		! Move gantry
		MoveAbsJ joints_end, v100, fine, tool0;

		! Read ending positions
		tcp_end_wobj0 := CRobT(\Tool:=tool0\WObj:=wobj0);
		tcp_end_floor := CRobT(\Tool:=tool0\WObj:=WobjFloor);

		TPWrite "End - Gantry: M1=" + NumToStr(joints_end.extax.eax_a, 1) + " M2=" + NumToStr(joints_end.extax.eax_b, 1) + " M3=" + NumToStr(joints_end.extax.eax_c, 1);

		! Calculate TCP changes
		wobj0_dx := tcp_end_wobj0.trans.x - tcp_start_wobj0.trans.x;
		wobj0_dy := tcp_end_wobj0.trans.y - tcp_start_wobj0.trans.y;
		wobj0_dz := tcp_end_wobj0.trans.z - tcp_start_wobj0.trans.z;

		floor_dx := tcp_end_floor.trans.x - tcp_start_floor.trans.x;
		floor_dy := tcp_end_floor.trans.y - tcp_start_floor.trans.y;
		floor_dz := tcp_end_floor.trans.z - tcp_start_floor.trans.z;

		! Save to file
		Open "HOME:/task2_gantry_test.txt", logfile \Append;
		Write logfile, "========================================";
		Write logfile, "TASK2 - Gantry Axis Movement Test (v1.4.0)";
		Write logfile, "Date: " + CDate() + " " + CTime();
		Write logfile, "========================================";
		WaitTime 0.05;
		Write logfile, "Gantry Joint Movement: M1=" + NumToStr(delta_m1, 1) + "mm, M2=" + NumToStr(delta_m2, 1) + "mm, M3=" + NumToStr(delta_m3, 1) + "mm";
		WaitTime 0.05;
		Write logfile, "wobj0 TCP moved: [" + NumToStr(wobj0_dx, 3) + ", " + NumToStr(wobj0_dy, 3) + ", " + NumToStr(wobj0_dz, 3) + "] mm";
		WaitTime 0.05;
		Write logfile, "Floor TCP moved: [" + NumToStr(floor_dx, 3) + ", " + NumToStr(floor_dy, 3) + ", " + NumToStr(floor_dz, 3) + "] mm";
		WaitTime 0.05;
		Write logfile, "========================================";
		Close logfile;

		TPWrite "Saved to: task2_gantry_test.txt";
	ENDPROC

	! ========================================
	! Quick Test - Gantry X Axis Movement
	! ========================================
	! Version: v1.4.1
	! Date: 2025-12-23
	! Purpose: Test M1DM3 (Gantry X) +1000mm movement from current position
	PROC TestGantryX()
		TPWrite "TASK2 - Gantry X Axis Test";
		TPWrite "Testing M1DM3 (X axis) +1000mm";
		TestGantryAxisMovement 1000, 0, 0;
		TPWrite "Test complete!";
	ENDPROC

	! ========================================
	! Quick Test - Gantry Y Axis Movement
	! ========================================
	PROC TestGantryY()
		TPWrite "TASK2 - Gantry Y Axis Test";
		TPWrite "Testing M2DM3 (Y axis) +500mm";
		TestGantryAxisMovement 0, 500, 0;
		TPWrite "Test complete!";
	ENDPROC

	! ========================================
	! Quick Test - Gantry Z Axis Movement
	! ========================================
	PROC TestGantryZ()
		TPWrite "TASK2 - Gantry Z Axis Test";
		TPWrite "Testing M3DM3 (Z axis) +200mm";
		TestGantryAxisMovement 0, 0, 200;
		TPWrite "Test complete!";
	ENDPROC

	! ========================================
	! Robot2 TCP Coordinate Test - XYZ Combined with Return
	! ========================================
	! Version: v1.5.0
	! Date: 2025-12-24
	! Purpose: Move Robot2 TCP in [X+50, Y+30, Z+20] from home position and return
	! MODE Selection (from /HOME/config.txt):
	!   MODE=0 (User's coordinate system):
	!     - Base: WobjFloor
	!     - Floor [+50, +30, +20] -> wobj0 [+50, +30, +20], Floor [+50, +30, +20]
	!   MODE=1 (Claude's coordinate system):
	!     - Base: wobj0
	!     - wobj0 [+50, +30, +20] -> Floor [+50, -30, -20]
	! Changes from v1.4.7:
	!   - Added config.txt MODE support
	!   - MODE=0: Use WobjFloor as base coordinate
	!   - MODE=1: Use wobj0 as base coordinate (default behavior)
	PROC TestRobot2_XYZ()
		VAR jointtarget original_pos;
		VAR jointtarget home_pos;
		VAR num config_mode;

		TPWrite "TASK2 - Robot2 Coordinate Test (v1.5.0)";

		! Read config mode
		config_mode := ReadConfigMode();
		TPWrite "Config MODE=" + NumToStr(config_mode, 0);

		! Save original joint position
		original_pos := CJointT();
		TPWrite "Original joint position saved";

		! Create home position (Robot2: [+90,0,0,0,30,0], keep gantry position)
		home_pos := original_pos;
		home_pos.robax.rax_1 := 90;
		home_pos.robax.rax_2 := 0;
		home_pos.robax.rax_3 := 0;
		home_pos.robax.rax_4 := 0;
		home_pos.robax.rax_5 := 30;
		home_pos.robax.rax_6 := 0;

		! Move to home position
		TPWrite "Moving to home position [+90,0,0,0,30,0]...";
		MoveAbsJ home_pos, v100, fine, tool0;
		TPWrite "At home position";

		! Perform coordinate test based on MODE
		IF config_mode = 0 THEN
			! MODE=0: User's coordinate - use WobjFloor as base
			TPWrite "MODE=0: Moving Floor: [+50, +30, +20]";
			TestCoordinateMovement 50, 30, 20, 0;
		ELSE
			! MODE=1: Claude's coordinate - use wobj0 as base
			TPWrite "MODE=1: Moving wobj0: [+50, +30, +20]";
			TestCoordinateMovement 50, 30, 20, 1;
		ENDIF

		! Return to original joint position
		TPWrite "Returning to original position...";
		MoveAbsJ original_pos, v100, fine, tool0;
		TPWrite "Returned to original position";

		TPWrite "Test complete! Check txt file";
	ENDPROC

	! ========================================
	! Update Robot1 Floor Position (local)
	! ========================================
	! Version: v1.5.2
	! Date: 2025-12-25
	! Purpose: Read Robot1 TCP from T_ROB1 without cross-task procedure call
	PROC UpdateRobot1FloorPositionLocal()
		robot1_floor_pos_t2 := CRobT(\TaskName:="T_ROB1"\Tool:=tool0\WObj:=WobjFloor);
	ENDPROC

	! ========================================
	! Set Robot2 Initial Position
	! ========================================
	! Version: v1.8.7
	! Date: 2026-01-05
	! Purpose: Move Robot2 to initial test position TCP [0, 488, -1000]
	! Position at R-axis center for easy calculation and verification
	! Uses WobjGantry_Rob2 which tracks current gantry position from TASK1
	! Changes in v1.8.7:
	!   - Use gantry extax from TASK1 when issuing MoveJ/MoveL targets
	! NOTE: This procedure does NOT control gantry (only TASK1 can control gantry)
	! Gantry should already be at HOME [0,0,0,0] by TASK1->SetRobot1InitialPosition
	! Version: v1.8.9
	! Date: 2026-01-05
	! Changes in v1.8.9:
	!   - Reduced TPWrite output and file logging to lower 41617 risk
	PROC SetRobot2InitialPosition()
		VAR jointtarget initial_joint;
		VAR jointtarget gantry_joint;
		VAR iodev logfile;

		! Open log file (summary logging)
		Open "HOME:/robot2_init_position.txt", logfile \Write;
		Write logfile, "Robot2 Init (" + TASK2_VERSION + ") Date=" + CDate() + " Time=" + CTime();

		! Step 1: Move Robot2 joints to intermediate position (tWeld2 HOME config)
		TPWrite "Robot2 init: Step1";
		initial_joint := CJointT();
		! Joint angles taught for tWeld2 HOME (confdata [0,0,0,4])
		initial_joint.robax.rax_1 := 0;
		initial_joint.robax.rax_2 := -48.88;
		initial_joint.robax.rax_3 := 6.22;
		initial_joint.robax.rax_4 := 0;
		initial_joint.robax.rax_5 := 8.26;
		initial_joint.robax.rax_6 := 0;
		! Keep current gantry position (DO NOT modify extax!)
		! extax values already set by CJointT()
		MoveAbsJ initial_joint, v100, fine, tool0;
		TPWrite "Robot2 init: Step1 done";
		Write logfile, "Step1 done (intermediate joint)";

		! v1.9.46: Step2 Cartesian refinement REMOVED
		! Robot2 is NOT gantry-configured - controller thinks base is fixed
		! At non-home gantry (especially R!=0), any Cartesian motion (MoveL/MoveJ)
		! converts WobjGantry_Rob2 target to world coords using fixed base -> 50050
		! Step1 MoveAbsJ already sets exact HOME joints - no refinement needed
		! Joint-space motion is gantry-position-independent (always works)

		! Log gantry position for reference
		gantry_joint := CJointT(\TaskName:="T_ROB1");
		Write logfile, "GantryPos from TASK1: X=" + NumToStr(gantry_joint.extax.eax_a,1)
			+ " Y=" + NumToStr(gantry_joint.extax.eax_b,1)
			+ " Z=" + NumToStr(gantry_joint.extax.eax_c,1)
			+ " R=" + NumToStr(gantry_joint.extax.eax_d,1);

		! Log current joint angles for verification
		initial_joint := CJointT();
		Write logfile, "Final joints: J1=" + NumToStr(initial_joint.robax.rax_1, 2)
			+ " J2=" + NumToStr(initial_joint.robax.rax_2, 2)
			+ " J3=" + NumToStr(initial_joint.robax.rax_3, 2)
			+ " J5=" + NumToStr(initial_joint.robax.rax_5, 2);

		TPWrite "Robot2 init: done";
		Write logfile, "Init done (joint-space only) at " + CTime();
		Close logfile;

		! Initialize robot2_floor_pos_t1 for cross-task measurement (v1.7.43)
		UpdateRobot2FloorPosition;
	ERROR
		TPWrite "ERROR in SetRobot2InitialPosition: " + NumToStr(ERRNO, 0);
		Close logfile;
		STOP;
	ENDPROC

	! ========================================
	! Log Current Position (for HOME teaching)
	! ========================================
	! Usage: Jog Robot2 to desired position -> Call from FlexPendant
	!        FlexPendant: ABB Menu -> Program Editor -> Debug -> Call Routine
	! Output: HOME:/current_position_r2.txt
	PROC LogCurrentPosition()
		VAR iodev logfile;
		VAR robtarget rt_tool0;
		VAR robtarget rt_tw2_wobj0;
		VAR robtarget rt_tw2_gantry;
		VAR jointtarget jt;

		Open "HOME:/current_position_r2.txt", logfile \Write;
		Write logfile, "=== ROB_2 Position Log " + CDate() + " " + CTime() + " ===";

		! --- JointTarget ---
		jt := CJointT();
		Write logfile, "";
		Write logfile, "--- ROB_2 JointTarget ---";
		Write logfile, "robax: [" + NumToStr(jt.robax.rax_1,3) + ", "
			+ NumToStr(jt.robax.rax_2,3) + ", " + NumToStr(jt.robax.rax_3,3) + ", "
			+ NumToStr(jt.robax.rax_4,3) + ", " + NumToStr(jt.robax.rax_5,3) + ", "
			+ NumToStr(jt.robax.rax_6,3) + "]";

		! --- RobTarget tool0/wobj0 ---
		rt_tool0 := CRobT(\Tool:=tool0\WObj:=wobj0);
		Write logfile, "";
		Write logfile, "--- ROB_2 RobTarget (tool0, wobj0) ---";
		Write logfile, "[[" + NumToStr(rt_tool0.trans.x,3) + ","
			+ NumToStr(rt_tool0.trans.y,3) + ","
			+ NumToStr(rt_tool0.trans.z,3) + "],["
			+ NumToStr(rt_tool0.rot.q1,5) + ","
			+ NumToStr(rt_tool0.rot.q2,5) + ","
			+ NumToStr(rt_tool0.rot.q3,5) + ","
			+ NumToStr(rt_tool0.rot.q4,5) + "],["
			+ NumToStr(rt_tool0.robconf.cf1,0) + ","
			+ NumToStr(rt_tool0.robconf.cf4,0) + ","
			+ NumToStr(rt_tool0.robconf.cf6,0) + ","
			+ NumToStr(rt_tool0.robconf.cfx,0) + "],extax]";

		! --- RobTarget tWeld2/wobj0 ---
		rt_tw2_wobj0 := CRobT(\Tool:=tWeld2\WObj:=wobj0);
		Write logfile, "";
		Write logfile, "--- ROB_2 RobTarget (tWeld2, wobj0) ---";
		Write logfile, "[[" + NumToStr(rt_tw2_wobj0.trans.x,3) + ","
			+ NumToStr(rt_tw2_wobj0.trans.y,3) + ","
			+ NumToStr(rt_tw2_wobj0.trans.z,3) + "],["
			+ NumToStr(rt_tw2_wobj0.rot.q1,5) + ","
			+ NumToStr(rt_tw2_wobj0.rot.q2,5) + ","
			+ NumToStr(rt_tw2_wobj0.rot.q3,5) + ","
			+ NumToStr(rt_tw2_wobj0.rot.q4,5) + "],["
			+ NumToStr(rt_tw2_wobj0.robconf.cf1,0) + ","
			+ NumToStr(rt_tw2_wobj0.robconf.cf4,0) + ","
			+ NumToStr(rt_tw2_wobj0.robconf.cf6,0) + ","
			+ NumToStr(rt_tw2_wobj0.robconf.cfx,0) + "],extax]";

		! --- RobTarget tWeld2/WobjGantry_Rob2 ---
		UpdateGantryWobj_Rob2;
		rt_tw2_gantry := CRobT(\Tool:=tWeld2\WObj:=WobjGantry_Rob2);
		Write logfile, "";
		Write logfile, "--- ROB_2 RobTarget (tWeld2, WobjGantry_Rob2) ---";
		Write logfile, "[[" + NumToStr(rt_tw2_gantry.trans.x,3) + ","
			+ NumToStr(rt_tw2_gantry.trans.y,3) + ","
			+ NumToStr(rt_tw2_gantry.trans.z,3) + "],["
			+ NumToStr(rt_tw2_gantry.rot.q1,5) + ","
			+ NumToStr(rt_tw2_gantry.rot.q2,5) + ","
			+ NumToStr(rt_tw2_gantry.rot.q3,5) + ","
			+ NumToStr(rt_tw2_gantry.rot.q4,5) + "],["
			+ NumToStr(rt_tw2_gantry.robconf.cf1,0) + ","
			+ NumToStr(rt_tw2_gantry.robconf.cf4,0) + ","
			+ NumToStr(rt_tw2_gantry.robconf.cf6,0) + ","
			+ NumToStr(rt_tw2_gantry.robconf.cfx,0) + "],extax]";

		Close logfile;
		TPWrite "ROB_2 position saved to HOME:/current_position_r2.txt";
	ENDPROC

	! ========================================
	! Set Robot2 TCP Offset for Mode2
	! ========================================
	! Version: v1.8.12
	! Date: 2026-01-06
	! Purpose: Move Robot2 TCP to offset using WobjGantry_Rob2
	! Changes in v1.8.39:
	!   - Use shared offsets from TASK1 (no config.txt read in TASK2)
	PROC SetRobot2OffsetPosition()
		VAR iodev diagfile;
		VAR jointtarget gantry_joint;
		VAR jointtarget task1_joints;  ! v1.8.69: For reading R angle from TASK1
		VAR jointtarget current_joints;  ! v1.8.70: For saving offset joints
		VAR robtarget offset_tcp;
		VAR num tcp_offset_x;
		VAR num tcp_offset_y;
		VAR num tcp_offset_z;
		VAR num wait_count;
		VAR num r_angle;
		VAR num calc_offset_x;
		VAR num calc_offset_y;

		! v1.8.75: Re-add MoveL for initial offset (50426 error fixed in system config)
		! - Initial call: MoveL to offset position using WobjGantry_Rob2
		! - Reposition call: Skip MoveL (joints maintained)

		Open "HOME:/task2_mode2_offset.txt", diagfile \Write;
		Write diagfile, "Mode2 Offset (" + TASK2_VERSION + ") Date=" + CDate() + " Time=" + CTime();

		IF mode2_r2_reposition_trigger THEN
			! ===== REPOSITION CALL =====
			! Gantry has moved, Robot2 joints stay at offset position (no motion needed)
			Write diagfile, "REPOSITION: Joints maintained (no motion)";
			mode2_r2_reposition_done := TRUE;
			TPWrite "R2: Reposition done (joints maintained)";
		ELSE
			! ===== INITIAL CALL =====
			! Move Robot2 TCP to offset position using MoveL
			Write diagfile, "INITIAL: MoveL to offset position";

			! Read offsets from PERS variables (set by TASK1)
			tcp_offset_x := mode2_r2_offset_x;
			tcp_offset_y := mode2_r2_offset_y;
			tcp_offset_z := mode2_r2_offset_z;
			Write diagfile, "Offsets: X=" + NumToStr(tcp_offset_x, 1) + " Y=" + NumToStr(tcp_offset_y, 1) + " Z=" + NumToStr(tcp_offset_z, 1);

			! Update WobjGantry_Rob2 to current gantry position
			UpdateGantryWobj_Rob2;
			gantry_joint := CJointT(\TaskName:="T_ROB1");
			Write diagfile, "WobjGantry_Rob2 updated, gantry extax read";

			! Calculate target position in WobjGantry_Rob2
			! Robot2 init position: [0, 488, -1000] in WobjGantry_Rob2
			! Offset: tcp_offset_y = -100 means 100mm toward Robot2 base
			! Target: [0, 488 + (-100), -1000] = [0, 388, -1000]
			calc_offset_x := tcp_offset_x;
			calc_offset_y := 488 + tcp_offset_y;  ! 488 + (-100) = 388
			Write diagfile, "Target: X=" + NumToStr(calc_offset_x, 1) + " Y=" + NumToStr(calc_offset_y, 1);

			offset_tcp := [[calc_offset_x, calc_offset_y, -1000 + tcp_offset_z],
			               [0.5, -0.5, -0.5, -0.5], [0, 0, 0, 0], gantry_joint.extax];
			Write diagfile, "Offset TCP: [" + NumToStr(offset_tcp.trans.x, 1) + ", "
			               + NumToStr(offset_tcp.trans.y, 1) + ", "
			               + NumToStr(offset_tcp.trans.z, 1) + "]";

			! MoveL to offset position (at HOME, this works)
			TPWrite "R2: MoveL to offset...";
			MoveL offset_tcp, v100, fine, tool0\WObj:=WobjGantry_Rob2;
			TPWrite "R2: MoveL done";
			Write diagfile, "MoveL completed";

			! Save offset joints for reposition calls
			current_joints := CJointT();
			robot2_offset_joints := current_joints.robax;
			Write diagfile, "Offset joints saved";

			! Note: mode2_r2_initial_offset_done is set in main() after config_ready wait
			! This prevents race condition with TASK1's flag reset
			Write diagfile, "MoveL and joint save complete (flag set by main)";
			TPWrite "R2: Offset position reached";
		ENDIF

		Close diagfile;

	ERROR
		Write diagfile, "ERROR in SetRobot2OffsetPosition: " + NumToStr(ERRNO, 0);
		Close diagfile;
		IF ERRNO = ERR_FILEOPEN THEN
			TPWrite "ERROR: Cannot open log file";
		ELSE
			TPWrite "ERROR in SetRobot2OffsetPosition: " + NumToStr(ERRNO, 0);
		ENDIF
		STOP;
	ENDPROC

	! ========================================
	! Update Robot2 Floor Position
	! ========================================
	! Version: v1.7.50
	! Date: 2025-12-31
	! Purpose: Placeholder - TASK1 calculates Robot2 Floor position
	! TASK1's UpdateRobot2BaseDynamicWobj() calculates robot2_floor_pos_t1 directly
	! TASK2 cannot sense gantry movement, so TASK1 does the calculation:
	!   1. TASK1 reads current gantry position
	!   2. TASK1 calculates Robot2 base Floor position
	!   3. TASK1 reads Robot2 TCP wobj0 using CRobT(\TaskName:="T_ROB2")
	!   4. TASK1 combines: robot2_floor_pos_t1 = base Floor + TCP wobj0
	! This procedure does nothing - robot2_floor_pos_t1 already updated by TASK1
	PROC UpdateRobot2FloorPosition()
		! Do nothing - TASK1's UpdateRobot2BaseDynamicWobj() already updated robot2_floor_pos_t1
		! This procedure kept for backward compatibility
		RETURN;
	ENDPROC

	! ========================================
	! Update Gantry Work Object for Robot2
	! ========================================
	! Version: v1.7.50
	! Date: 2025-12-31
	! Purpose: Update WobjGantry_Rob2 to reflect current gantry position and rotation
	! Robot2 cannot control gantry - must read position from TASK1
	! This allows Robot2 TCP control in Floor coordinates regardless of gantry position
	! R-axis orientation: R=0 means gantry parallel to Y-axis (Floor coordinate)
	! Must be called before using WobjGantry_Rob2 for TCP movements
	PROC UpdateGantryWobj_Rob2()
		VAR jointtarget current_gantry;
		VAR num r_deg;

		! Read current gantry position from TASK1 (Robot2 cannot sense this directly)
		current_gantry := CJointT(\TaskName:="T_ROB1");

		! Update WobjGantry_Rob2 position to current gantry location
		WobjGantry_Rob2.uframe.trans.x := current_gantry.extax.eax_a;
		WobjGantry_Rob2.uframe.trans.y := current_gantry.extax.eax_b;
		WobjGantry_Rob2.uframe.trans.z := current_gantry.extax.eax_c;

		! WobjGantry_Rob2 orientation
		! IMPORTANT: WobjGantry_Rob2 coordinate system is always aligned with World/Floor
		! R-axis rotation affects robot base, NOT work object orientation
		! Robot2 base is physically rotated 90deg, but work object remains aligned with World
		! Keep quaternion as identity (no rotation)
		WobjGantry_Rob2.uframe.rot.q1 := 1;
		WobjGantry_Rob2.uframe.rot.q2 := 0;
		WobjGantry_Rob2.uframe.rot.q3 := 0;
		WobjGantry_Rob2.uframe.rot.q4 := 0;

		r_deg := current_gantry.extax.eax_d;

		TPWrite "WobjGantry_Rob2 updated: [" + NumToStr(current_gantry.extax.eax_a,0) + ", "
		                                    + NumToStr(current_gantry.extax.eax_b,0) + ", "
		                                    + NumToStr(current_gantry.extax.eax_c,0) + ", R="
		                                    + NumToStr(r_deg,1) + "]";
	ENDPROC

	! ========================================
	! Calculate Robot Distance
	! ========================================
	! Version: v1.5.1
	! Date: 2025-12-25
	! Purpose: Calculate 3D distance between Robot1 and Robot2 in Floor coordinate
	! Returns: Distance in mm
	FUNC num CalculateRobotDistance()
		VAR num dx;
		VAR num dy;
		VAR num dz;

		dx := robot2_floor_pos_t1.trans.x - robot1_floor_pos_t2.trans.x;
		dy := robot2_floor_pos_t1.trans.y - robot1_floor_pos_t2.trans.y;
		dz := robot2_floor_pos_t1.trans.z - robot1_floor_pos_t2.trans.z;

		RETURN Sqrt(Pow(dx, 2) + Pow(dy, 2) + Pow(dz, 2));
	ENDFUNC

	! ========================================
	! Measure Robot Distance
	! ========================================
	! Version: v1.5.1
	! Date: 2025-12-25
	! Purpose: Measure and log distance between Robot1 and Robot2
	! Output: TP display + /HOME/robot_distance_log.txt
	PROC MeasureRobotDistance()
		VAR num distance;
		VAR iodev logfile;

		TPWrite "========================================";
		TPWrite "Robot Distance Measurement (v1.5.1)";
		TPWrite "========================================";

		! Update both robot positions
		UpdateRobot1FloorPositionLocal;
		UpdateRobot2FloorPosition;

		! Calculate distance
		distance := CalculateRobotDistance();

		! Display on TP
		TPWrite "Robot1 Floor Position:";
		TPWrite "  X = " + NumToStr(robot1_floor_pos_t2.trans.x, 2) + " mm";
		TPWrite "  Y = " + NumToStr(robot1_floor_pos_t2.trans.y, 2) + " mm";
		TPWrite "  Z = " + NumToStr(robot1_floor_pos_t2.trans.z, 2) + " mm";
		TPWrite "";
		TPWrite "Robot2 Floor Position:";
		TPWrite "  X = " + NumToStr(robot2_floor_pos_t1.trans.x, 2) + " mm";
		TPWrite "  Y = " + NumToStr(robot2_floor_pos_t1.trans.y, 2) + " mm";
		TPWrite "  Z = " + NumToStr(robot2_floor_pos_t1.trans.z, 2) + " mm";
		TPWrite "";
		TPWrite "Distance between robots: " + NumToStr(distance, 2) + " mm";
		TPWrite "========================================";

		! Save to log file
		Open "HOME:/robot_distance_log.txt", logfile \Write;

		Write logfile, "========================================";
		Write logfile, "Robot Distance Measurement (v1.5.1)";
		Write logfile, "========================================";
		Write logfile, "Date: " + CDate();
		Write logfile, "Time: " + CTime();
		Write logfile, "";
		Write logfile, "Robot1 Floor Position (tool0):";
		Write logfile, "  X = " + NumToStr(robot1_floor_pos_t2.trans.x, 2) + " mm";
		Write logfile, "  Y = " + NumToStr(robot1_floor_pos_t2.trans.y, 2) + " mm";
		Write logfile, "  Z = " + NumToStr(robot1_floor_pos_t2.trans.z, 2) + " mm";
		Write logfile, "";
		Write logfile, "Robot2 Floor Position (tool0):";
		Write logfile, "  X = " + NumToStr(robot2_floor_pos_t1.trans.x, 2) + " mm";
		Write logfile, "  Y = " + NumToStr(robot2_floor_pos_t1.trans.y, 2) + " mm";
		Write logfile, "  Z = " + NumToStr(robot2_floor_pos_t1.trans.z, 2) + " mm";
		Write logfile, "";
		Write logfile, "Distance: " + NumToStr(distance, 2) + " mm";
		Write logfile, "========================================\0A";

		Close logfile;
		TPWrite "Saved to: /HOME/robot_distance_log.txt";

	ERROR
		TPWrite "ERROR in MeasureRobotDistance: " + NumToStr(ERRNO, 0);
		Close logfile;
		TRYNEXT;
	ENDPROC

	! ========================================
	! Test Robot2 Base Height
	! ========================================
	! Version: v1.7.14
	! Date: 2025-12-28
	! Purpose: Check tool0 TCP height from base at specific joint angles
	! Uses WobjFloor_Rob2
	! Output: TP display + /HOME/robot2_base_height.txt
	PROC TestRobot2BaseHeight()
		VAR jointtarget test_pos;
		VAR robtarget tcp_wobj0;
		VAR robtarget tcp_floor;
		VAR iodev logfile;

		TPWrite "========================================";
		TPWrite "Robot2 Base Height Test (v1.7.14)";

		! Get current position
		test_pos := CJointT();

		! Set robot joints to [+90, 0, 0, 0, 0, 0]
		test_pos.robax.rax_1 := 90;
		test_pos.robax.rax_2 := 0;
		test_pos.robax.rax_3 := 0;
		test_pos.robax.rax_4 := 0;
		test_pos.robax.rax_5 := 0;
		test_pos.robax.rax_6 := 0;

		! Move to test position
		TPWrite "Moving to test position [+90,0,0,0,0,0]...";
		MoveAbsJ test_pos, v100, fine, tool0;
		WaitTime 0.5;

		! Read TCP position in wobj0
		tcp_wobj0 := CRobT(\Tool:=tool0\WObj:=wobj0);

		! Read TCP position in Floor coordinate (using Robot2-specific Floor)
		tcp_floor := CRobT(\Tool:=tool0\WObj:=WobjFloor_Rob2);

		! Display on TP
		TPWrite "Robot2 wobj0:";
		TPWrite "  X = " + NumToStr(tcp_wobj0.trans.x, 2);
		TPWrite "  Y = " + NumToStr(tcp_wobj0.trans.y, 2);
		TPWrite "  Z = " + NumToStr(tcp_wobj0.trans.z, 2);

		TPWrite "Robot2 Floor (WobjFloor_Rob2):";
		TPWrite "  X = " + NumToStr(tcp_floor.trans.x, 2);
		TPWrite "  Y = " + NumToStr(tcp_floor.trans.y, 2);
		TPWrite "  Z = " + NumToStr(tcp_floor.trans.z, 2);

		TPWrite "========================================";

		! Save to log file
		Open "HOME:/robot2_base_height.txt", logfile \Write;

		Write logfile, "========================================";
		Write logfile, "Robot2 Base Height Test (v1.7.14)";
		Write logfile, "========================================";
		Write logfile, "Date: " + CDate();
		Write logfile, "Time: " + CTime();
		Write logfile, "";
		Write logfile, "Joint Angles: [+90, 0, 0, 0, 0, 0]";
		Write logfile, "";
		Write logfile, "Robot2 wobj0 (tool0):";
		Write logfile, "  X = " + NumToStr(tcp_wobj0.trans.x, 2) + " mm";
		Write logfile, "  Y = " + NumToStr(tcp_wobj0.trans.y, 2) + " mm";
		Write logfile, "  Z = " + NumToStr(tcp_wobj0.trans.z, 2) + " mm";
		Write logfile, "";
		Write logfile, "Robot2 Floor (tool0) - using WobjFloor_Rob2:";
		Write logfile, "  X = " + NumToStr(tcp_floor.trans.x, 2) + " mm";
		Write logfile, "  Y = " + NumToStr(tcp_floor.trans.y, 2) + " mm";
		Write logfile, "  Z = " + NumToStr(tcp_floor.trans.z, 2) + " mm";
		Write logfile, "========================================\0A";

		Close logfile;
		TPWrite "Saved to: /HOME/robot2_base_height.txt";

	ERROR
		TPWrite "ERROR in TestRobot2BaseHeight: " + NumToStr(ERRNO, 0);
		Close logfile;
		TRYNEXT;
	ENDPROC

	! ========================================
	! Test Gantry Movement Effect on Floor Coordinates
	! ========================================
	! Version: v1.7.29
	! Date: 2025-12-29
	! Purpose: Test if Floor coordinates change when gantry moves
	! Reads gantry movement from config.txt (X, Y, Z, R)
	! Initial position: Robot1 [-90,0,0,0,0,0], Robot2 [+90,0,0,0,0,0]
	! Gantry HOME: [-9500, 5300, 700, 0] (safe Z position, max=1000mm)
	! Gantry moved: HOME + config offset
	! Note: Based on 12-23 backup fnCoordToJoint function
	! Output: /HOME/gantry_floor_test.txt
	PROC TestGantryFloorCoordinates()
		VAR jointtarget rob1_init;
		VAR jointtarget rob2_init;
		VAR jointtarget home_pos;
		VAR jointtarget moved_pos;
		VAR robtarget rob1_floor_before;
		VAR robtarget rob2_floor_before;
		VAR robtarget rob1_floor_after;
		VAR robtarget rob2_floor_after;
		VAR iodev logfile;
		VAR iodev configfile;
		VAR string line;
		VAR string value_str;
		VAR bool found_value;
		VAR bool found_x;
		VAR bool found_y;
		VAR bool found_z;
		VAR bool found_r;
		VAR num gantry_x_offset;
		VAR num gantry_y_offset;
		VAR num gantry_z_offset;
		VAR num gantry_r_offset;

		TPWrite "========================================";
		TPWrite "Gantry Floor Test (v1.7.28)";

		! Initialize variables
		gantry_x_offset := 0;
		gantry_y_offset := 0;
		gantry_z_offset := 0;
		gantry_r_offset := 0;

		! Check Robot1 position
		TPWrite "Checking Robot1 position...";
		rob1_init := CJointT(\TaskName:="T_ROB1");
		IF Abs(rob1_init.robax.rax_1 + 90) > 5 THEN
			TPWrite "WARNING: Robot1 is NOT at initial position!";
			TPWrite "Current Robot1 J1: " + NumToStr(rob1_init.robax.rax_1, 1);
			TPWrite "Expected: -90 degrees";
			TPWrite "Please run TASK1->SetRobot1InitialPosition first";
			TPWrite "Then re-run this test";
			STOP;
		ENDIF
		TPWrite "Robot1 position OK (J1=-90)";

		! Move Robot2 to initial test position (keep current gantry position)
		TPWrite "Moving Robot2 to initial position...";
		rob2_init := CJointT();
		! Set robot joints only
		rob2_init.robax.rax_1 := 90;
		rob2_init.robax.rax_2 := 0;
		rob2_init.robax.rax_3 := 0;
		rob2_init.robax.rax_4 := 0;
		rob2_init.robax.rax_5 := 0;
		rob2_init.robax.rax_6 := 0;
		! Keep current gantry position (DO NOT force to 0)
		! extax values already set by CJointT()
		MoveAbsJ rob2_init, v100, fine, tool0;
		TPWrite "Robot2 initial position reached!";

		! Now move gantry to HOME position
		TPWrite "Moving gantry to HOME position...";
		home_pos := rob2_init;
		home_pos.extax.eax_a := -9500;  ! X1 = WobjFloor origin X
		home_pos.extax.eax_b := 5300;   ! Y = WobjFloor origin Y
		home_pos.extax.eax_c := 700;    ! Z = Safe mid-height (max=1000, ref: 12-23 backup)
		home_pos.extax.eax_d := 0;      ! R = 0
		! eax_e: keep from CJointT() (not used)
		home_pos.extax.eax_f := -9500;  ! X2 = X1 (Master-Follower sync!)
		MoveAbsJ home_pos, v100, fine, tool0;
		TPWrite "Gantry at HOME position (WobjFloor origin)";
		TPWrite "Both robots ready!";

		! Read gantry offsets from config.txt (simple approach)
		TPWrite "Opening config.txt...";
		Open "HOME:/config.txt", configfile \Read;
		TPWrite "Reading config values...";

		! Read GANTRY_X
		found_x := FALSE;
		WHILE found_x = FALSE DO
			line := ReadStr(configfile \RemoveCR);
			IF StrFind(line, 1, "GANTRY_X=") = 1 THEN
				IF StrLen(line) >= 10 THEN
					value_str := StrPart(line, 10, StrLen(line) - 9);
					found_value := StrToVal(value_str, gantry_x_offset);
					found_x := TRUE;
					TPWrite "Found GANTRY_X=" + NumToStr(gantry_x_offset, 0);
				ENDIF
			ENDIF
		ENDWHILE

		! Read GANTRY_Y
		found_y := FALSE;
		WHILE found_y = FALSE DO
			line := ReadStr(configfile \RemoveCR);
			IF StrFind(line, 1, "GANTRY_Y=") = 1 THEN
				IF StrLen(line) >= 10 THEN
					value_str := StrPart(line, 10, StrLen(line) - 9);
					found_value := StrToVal(value_str, gantry_y_offset);
					found_y := TRUE;
					TPWrite "Found GANTRY_Y=" + NumToStr(gantry_y_offset, 0);
				ENDIF
			ENDIF
		ENDWHILE

		! Read GANTRY_Z
		found_z := FALSE;
		WHILE found_z = FALSE DO
			line := ReadStr(configfile \RemoveCR);
			IF StrFind(line, 1, "GANTRY_Z=") = 1 THEN
				IF StrLen(line) >= 10 THEN
					value_str := StrPart(line, 10, StrLen(line) - 9);
					found_value := StrToVal(value_str, gantry_z_offset);
					found_z := TRUE;
					TPWrite "Found GANTRY_Z=" + NumToStr(gantry_z_offset, 0);
				ENDIF
			ENDIF
		ENDWHILE

		! Read GANTRY_R
		found_r := FALSE;
		WHILE found_r = FALSE DO
			line := ReadStr(configfile \RemoveCR);
			IF StrFind(line, 1, "GANTRY_R=") = 1 THEN
				IF StrLen(line) >= 10 THEN
					value_str := StrPart(line, 10, StrLen(line) - 9);
					found_value := StrToVal(value_str, gantry_r_offset);
					found_r := TRUE;
					TPWrite "Found GANTRY_R=" + NumToStr(gantry_r_offset, 1);
				ENDIF
			ENDIF
		ENDWHILE

		Close configfile;
		TPWrite "Config reading complete!";

		TPWrite "Gantry offsets:";
		TPWrite "  X=" + NumToStr(gantry_x_offset, 0) + " mm";
		TPWrite "  Y=" + NumToStr(gantry_y_offset, 0) + " mm";
		TPWrite "  Z=" + NumToStr(gantry_z_offset, 0) + " mm";
		TPWrite "  R=" + NumToStr(gantry_r_offset, 1) + " deg";

		! Move to HOME position (all gantry axes = 0)
		TPWrite "Moving to HOME position...";
		home_pos := CJointT();
		home_pos.extax.eax_a := 0;  ! X axis
		home_pos.extax.eax_b := 0;  ! Y axis
		home_pos.extax.eax_c := 0;  ! Z axis
		home_pos.extax.eax_d := 0;  ! R axis
		MoveAbsJ home_pos, v100, fine, tool0;
		WaitTime 1.0;

		! Measure BEFORE gantry movement
		TPWrite "Measuring before gantry move...";
		UpdateRobot1FloorPositionLocal;
		UpdateRobot2FloorPosition;
		rob1_floor_before := robot1_floor_pos_t2;
		rob2_floor_before := robot2_floor_pos_t1;

		! Move gantry axes (HOME + offset)
		TPWrite "Moving gantry...";
		moved_pos := home_pos;
		moved_pos.extax.eax_a := -9500 + gantry_x_offset;  ! X1 = HOME + offset
		moved_pos.extax.eax_b := 5300 + gantry_y_offset;   ! Y = HOME + offset
		moved_pos.extax.eax_c := 700 + gantry_z_offset;    ! Z = HOME + offset (max=1000)
		moved_pos.extax.eax_d := 0 + gantry_r_offset;      ! R = HOME + offset
		! eax_e: keep from home_pos/CJointT() (not used)
		moved_pos.extax.eax_f := -9500 + gantry_x_offset;  ! X2 = X1 (Master-Follower sync!)
		MoveAbsJ moved_pos, v100, fine, tool0;
		WaitTime 1.0;

		! Measure AFTER gantry movement
		TPWrite "Measuring after gantry move...";
		UpdateRobot1FloorPositionLocal;
		UpdateRobot2FloorPosition;
		rob1_floor_after := robot1_floor_pos_t2;
		rob2_floor_after := robot2_floor_pos_t1;

		! Return to HOME position
		TPWrite "Returning to HOME position...";
		MoveAbsJ home_pos, v100, fine, tool0;

		! Save results
		Open "HOME:/gantry_floor_test.txt", logfile \Write;

		Write logfile, "========================================";
		Write logfile, "Gantry Floor Coordinate Test (v1.7.29)";
		Write logfile, "========================================";
		Write logfile, "Date: " + CDate();
		Write logfile, "Time: " + CTime();
		Write logfile, "";
		Write logfile, "HOME Position (WobjFloor origin):";
		Write logfile, "  Gantry: X1=-9500, Y=5300, Z=2100, R=0, X2=-9500";
		Write logfile, "";
		Write logfile, "Initial Position:";
		Write logfile, "  Robot1: [-90,0,0,0,0,0]";
		Write logfile, "  Robot2: [+90,0,0,0,0,0]";
		Write logfile, "  Gantry: at HOME (WobjFloor origin)";
		Write logfile, "";
		Write logfile, "Gantry Movement:";
		Write logfile, "  X = " + NumToStr(gantry_x_offset, 2) + " mm (X1 and X2 synchronized)";
		Write logfile, "  Y = " + NumToStr(gantry_y_offset, 2) + " mm";
		Write logfile, "  Z = " + NumToStr(gantry_z_offset, 2) + " mm";
		Write logfile, "  R = " + NumToStr(gantry_r_offset, 2) + " deg";
		Write logfile, "";
		Write logfile, "BEFORE Gantry Movement:";
		Write logfile, "------------------------";
		Write logfile, "Robot1 Floor (tool0):";
		Write logfile, "  X = " + NumToStr(rob1_floor_before.trans.x, 2) + " mm";
		Write logfile, "  Y = " + NumToStr(rob1_floor_before.trans.y, 2) + " mm";
		Write logfile, "  Z = " + NumToStr(rob1_floor_before.trans.z, 2) + " mm";
		Write logfile, "";
		Write logfile, "Robot2 Floor (tool0):";
		Write logfile, "  X = " + NumToStr(rob2_floor_before.trans.x, 2) + " mm";
		Write logfile, "  Y = " + NumToStr(rob2_floor_before.trans.y, 2) + " mm";
		Write logfile, "  Z = " + NumToStr(rob2_floor_before.trans.z, 2) + " mm";
		Write logfile, "";
		Write logfile, "AFTER Gantry Movement:";
		Write logfile, "----------------------";
		Write logfile, "Robot1 Floor (tool0):";
		Write logfile, "  X = " + NumToStr(rob1_floor_after.trans.x, 2) + " mm";
		Write logfile, "  Y = " + NumToStr(rob1_floor_after.trans.y, 2) + " mm";
		Write logfile, "  Z = " + NumToStr(rob1_floor_after.trans.z, 2) + " mm";
		Write logfile, "";
		Write logfile, "Robot2 Floor (tool0):";
		Write logfile, "  X = " + NumToStr(rob2_floor_after.trans.x, 2) + " mm";
		Write logfile, "  Y = " + NumToStr(rob2_floor_after.trans.y, 2) + " mm";
		Write logfile, "  Z = " + NumToStr(rob2_floor_after.trans.z, 2) + " mm";
		Write logfile, "";
		Write logfile, "DIFFERENCE:";
		Write logfile, "-----------";
		Write logfile, "Robot1 Floor Delta:";
		Write logfile, "  dX = " + NumToStr(rob1_floor_after.trans.x - rob1_floor_before.trans.x, 2) + " mm";
		Write logfile, "  dY = " + NumToStr(rob1_floor_after.trans.y - rob1_floor_before.trans.y, 2) + " mm";
		Write logfile, "  dZ = " + NumToStr(rob1_floor_after.trans.z - rob1_floor_before.trans.z, 2) + " mm";
		Write logfile, "";
		Write logfile, "Robot2 Floor Delta:";
		Write logfile, "  dX = " + NumToStr(rob2_floor_after.trans.x - rob2_floor_before.trans.x, 2) + " mm";
		Write logfile, "  dY = " + NumToStr(rob2_floor_after.trans.y - rob2_floor_before.trans.y, 2) + " mm";
		Write logfile, "  dZ = " + NumToStr(rob2_floor_after.trans.z - rob2_floor_before.trans.z, 2) + " mm";
		Write logfile, "========================================\0A";

		Close logfile;
		TPWrite "Saved to: /HOME/gantry_floor_test.txt";
		TPWrite "Test complete!";

	ERROR
		IF ERRNO = ERR_FILEOPEN THEN
			TPWrite "ERROR: Cannot open config.txt";
			STOP;
		ELSEIF ERRNO = ERR_FILEACC THEN
			TPWrite "ERROR: End of file or access error";
			TPWrite "Check config.txt format";
			Close configfile;
			STOP;
		ELSE
			TPWrite "ERROR in TestGantryFloorCoordinates";
			TPWrite "ERRNO: " + NumToStr(ERRNO, 0);
			Close logfile;
			Close configfile;
			STOP;
		ENDIF
	ENDPROC

! ========================================
! Weld Sequence Procedures (v1.9.0)
! ========================================
! Purpose: Robot2 weld sequence synchronization with TASK1
! Robot2 waits for TASK1 signal, then moves to weld position

! ----------------------------------------
! Robot2 Weld Ready - Wait and Move (2-step approach)
! ----------------------------------------
! v1.9.19: Step1 - MoveAbsJ to safe joint position
!          Step2 - MoveJ to wobj0 target position
PROC Robot2_WeldReady()
	VAR robtarget weld_target;
	VAR jointtarget safe_jt;

	TPWrite "[R2_WELD] Robot2 weld ready procedure started";
	TPWrite "[R2_WELD] Waiting for TASK1 weld start signal...";

	! Wait for TASK1 weld start signal
	WHILE NOT t1_weld_start DO
		WaitTime 0.1;
	ENDWHILE

	TPWrite "[R2_WELD] Received weld start signal from TASK1";

	! Step 1: Move to safe JOINT position first
	! Robot joints: [0, -10, -50, 0, -30, 0]
	safe_jt := CJointT();
	safe_jt.robax.rax_1 := 0;
	safe_jt.robax.rax_2 := -10;
	safe_jt.robax.rax_3 := -50;
	safe_jt.robax.rax_4 := 0;
	safe_jt.robax.rax_5 := -30;
	safe_jt.robax.rax_6 := 0;
	! Robot2 has no external axes
	safe_jt.extax.eax_a := 9E9;
	safe_jt.extax.eax_b := 9E9;
	safe_jt.extax.eax_c := 9E9;
	safe_jt.extax.eax_d := 9E9;
	safe_jt.extax.eax_e := 9E9;
	safe_jt.extax.eax_f := 9E9;
	TPWrite "[R2_WELD] Step1: MoveAbsJ to safe joints";
	MoveAbsJ safe_jt, v100, fine, tool0;

	! Step 2: Move to wobj0 target position
	! wobj0 target: [0, 118, -1300]
	weld_target.trans.x := 0;
	weld_target.trans.y := 118;
	weld_target.trans.z := -1300;
	weld_target.rot.q1 := WELD_R2_ORIENT_Q1;
	weld_target.rot.q2 := WELD_R2_ORIENT_Q2;
	weld_target.rot.q3 := WELD_R2_ORIENT_Q3;
	weld_target.rot.q4 := WELD_R2_ORIENT_Q4;
	weld_target.robconf.cf1 := 0;
	weld_target.robconf.cf4 := 0;
	weld_target.robconf.cf6 := 0;
	weld_target.robconf.cfx := 0;
	weld_target.extax.eax_a := 9E9;
	weld_target.extax.eax_b := 9E9;
	weld_target.extax.eax_c := 9E9;
	weld_target.extax.eax_d := 9E9;
	weld_target.extax.eax_e := 9E9;
	weld_target.extax.eax_f := 9E9;

	TPWrite "[R2_WELD] Step2: MoveJ to wobj0 [0, 118, -1300]";
	MoveJ weld_target, v100, fine, tool0\WObj:=wobj0;

	! Signal ready to TASK1
	t2_weld_ready := TRUE;

	TPWrite "[R2_WELD] Robot2 at weld position, signaled ready";
ENDPROC

! ----------------------------------------
! Robot2 Weld Hold - Maintain Position
! ----------------------------------------
! Maintains weld posture while TASK1 moves gantry
! Called after Robot2_WeldReady completes
PROC Robot2_WeldHold()
	TPWrite "[R2_WELD] Robot2 holding weld position...";

	! Wait for TASK1 weld complete signal
	WHILE NOT t1_weld_done DO
		WaitTime 0.1;
	ENDWHILE

	TPWrite "[R2_WELD] TASK1 weld complete, Robot2 released";
ENDPROC

! ----------------------------------------
! Robot2 Weld Sequence (Combined)
! ----------------------------------------
! Combined sequence: wait for signal, move to position, hold until done
PROC Robot2_WeldSequence()
	TPWrite "========================================";
	TPWrite "[R2_WELD] v1.9.0 Robot2 Weld Sequence Start";
	TPWrite "========================================";

	! Reset ready flag
	t2_weld_ready := FALSE;

	! Wait for signal and move to weld position
	Robot2_WeldReady;

	! Hold position until welding complete
	Robot2_WeldHold;

	TPWrite "========================================";
	TPWrite "[R2_WELD] Robot2 Weld Sequence Complete!";
	TPWrite "========================================";
ENDPROC

! ========================================
! Edge-based Weld Sequence (v2.0.0)
! ========================================
! Ported from PlanA - waits for TASK1 to position gantry,
! then moves Robot2 to weld position considering bRobSwap

! ----------------------------------------
! Robot2 Edge-based Weld Sequence (v1.9.37)
! ----------------------------------------
! Waits for t1_weld_position_ready, then positions Robot2
! v1.9.37: Weld tracking with position logging, edge data from TASK1
PROC Robot2_EdgeWeldSequence()
    ! ========================================
    ! Robot2 Edge Weld Sequence (v3.0.0)
    ! Ported from PlanA rWeld012()
    ! Uses Welds2{} + wobjWeldLine2 + fCalcWeldingpos()
    ! Simulation mode: MoveL (WELD_ARC_ENABLED=FALSE)
    ! ========================================
    VAR num nTempMmps;
    VAR num nHoldWeldVel;
    VAR jointtarget jCurrent;
    VAR iodev weld2_errlog;
    VAR num nErrorCount;
    VAR num nMotionErrorCount;

    TPWrite "[R2_WELD] Robot2_EdgeWeldSequence v4.0 start";
    nHoldWeldVel:=0.01;

    ! Signal TASK1 we are ready (unblocks Step 7 wait in Full Weld Sequence)
    t2_weld_ready := TRUE;

    ! --- Setup weld data (wd1..wd40) ---
    wd1:=[Welds2{1}.cpm/6,0,[5,0,Welds2{1}.voltage,Welds2{1}.wfs,0,Welds2{1}.Current,0,0,0],[0,0,0,0,0,0,0,0,0]];
    wd2:=[Welds2{2}.cpm/6,0,[5,0,Welds2{2}.voltage,Welds2{2}.wfs,0,Welds2{2}.Current,0,0,0],[0,0,0,0,0,0,0,0,0]];
    wd3:=[Welds2{3}.cpm/6,0,[5,0,Welds2{3}.voltage,Welds2{3}.wfs,0,Welds2{3}.Current,0,0,0],[0,0,0,0,0,0,0,0,0]];
    wd4:=[Welds2{4}.cpm/6,0,[5,0,Welds2{4}.voltage,Welds2{4}.wfs,0,Welds2{4}.Current,0,0,0],[0,0,0,0,0,0,0,0,0]];
    wd5:=[Welds2{5}.cpm/6,0,[5,0,Welds2{5}.voltage,Welds2{5}.wfs,0,Welds2{5}.Current,0,0,0],[0,0,0,0,0,0,0,0,0]];
    wd6:=[Welds2{6}.cpm/6,0,[5,0,Welds2{6}.voltage,Welds2{6}.wfs,0,Welds2{6}.Current,0,0,0],[0,0,0,0,0,0,0,0,0]];
    wd7:=[Welds2{7}.cpm/6,0,[5,0,Welds2{7}.voltage,Welds2{7}.wfs,0,Welds2{7}.Current,0,0,0],[0,0,0,0,0,0,0,0,0]];
    wd8:=[Welds2{8}.cpm/6,0,[5,0,Welds2{8}.voltage,Welds2{8}.wfs,0,Welds2{8}.Current,0,0,0],[0,0,0,0,0,0,0,0,0]];
    wd9:=[Welds2{9}.cpm/6,0,[5,0,Welds2{9}.voltage,Welds2{9}.wfs,0,Welds2{9}.Current,0,0,0],[0,0,0,0,0,0,0,0,0]];
    wd10:=[Welds2{10}.cpm/6,0,[5,0,Welds2{10}.voltage,Welds2{10}.wfs,0,Welds2{10}.Current,0,0,0],[0,0,0,0,0,0,0,0,0]];
    wd11:=[Welds2{11}.cpm/6,0,[5,0,Welds2{11}.voltage,Welds2{11}.wfs,0,Welds2{11}.Current,0,0,0],[0,0,0,0,0,0,0,0,0]];
    wd12:=[Welds2{12}.cpm/6,0,[5,0,Welds2{12}.voltage,Welds2{12}.wfs,0,Welds2{12}.Current,0,0,0],[0,0,0,0,0,0,0,0,0]];
    wd13:=[Welds2{13}.cpm/6,0,[5,0,Welds2{13}.voltage,Welds2{13}.wfs,0,Welds2{13}.Current,0,0,0],[0,0,0,0,0,0,0,0,0]];
    wd14:=[Welds2{14}.cpm/6,0,[5,0,Welds2{14}.voltage,Welds2{14}.wfs,0,Welds2{14}.Current,0,0,0],[0,0,0,0,0,0,0,0,0]];
    wd15:=[Welds2{15}.cpm/6,0,[5,0,Welds2{15}.voltage,Welds2{15}.wfs,0,Welds2{15}.Current,0,0,0],[0,0,0,0,0,0,0,0,0]];
    wd16:=[Welds2{16}.cpm/6,0,[5,0,Welds2{16}.voltage,Welds2{16}.wfs,0,Welds2{16}.Current,0,0,0],[0,0,0,0,0,0,0,0,0]];
    wd17:=[Welds2{17}.cpm/6,0,[5,0,Welds2{17}.voltage,Welds2{17}.wfs,0,Welds2{17}.Current,0,0,0],[0,0,0,0,0,0,0,0,0]];
    wd18:=[Welds2{18}.cpm/6,0,[5,0,Welds2{18}.voltage,Welds2{18}.wfs,0,Welds2{18}.Current,0,0,0],[0,0,0,0,0,0,0,0,0]];
    wd19:=[Welds2{19}.cpm/6,0,[5,0,Welds2{19}.voltage,Welds2{19}.wfs,0,Welds2{19}.Current,0,0,0],[0,0,0,0,0,0,0,0,0]];
    wd20:=[Welds2{20}.cpm/6,0,[5,0,Welds2{20}.voltage,Welds2{20}.wfs,0,Welds2{20}.Current,0,0,0],[0,0,0,0,0,0,0,0,0]];
    wd21:=[Welds2{21}.cpm/6,0,[5,0,Welds2{21}.voltage,Welds2{21}.wfs,0,Welds2{21}.Current,0,0,0],[0,0,0,0,0,0,0,0,0]];
    wd22:=[Welds2{22}.cpm/6,0,[5,0,Welds2{22}.voltage,Welds2{22}.wfs,0,Welds2{22}.Current,0,0,0],[0,0,0,0,0,0,0,0,0]];
    wd23:=[Welds2{23}.cpm/6,0,[5,0,Welds2{23}.voltage,Welds2{23}.wfs,0,Welds2{23}.Current,0,0,0],[0,0,0,0,0,0,0,0,0]];
    wd24:=[Welds2{24}.cpm/6,0,[5,0,Welds2{24}.voltage,Welds2{24}.wfs,0,Welds2{24}.Current,0,0,0],[0,0,0,0,0,0,0,0,0]];
    wd25:=[Welds2{25}.cpm/6,0,[5,0,Welds2{25}.voltage,Welds2{25}.wfs,0,Welds2{25}.Current,0,0,0],[0,0,0,0,0,0,0,0,0]];
    wd26:=[Welds2{26}.cpm/6,0,[5,0,Welds2{26}.voltage,Welds2{26}.wfs,0,Welds2{26}.Current,0,0,0],[0,0,0,0,0,0,0,0,0]];
    wd27:=[Welds2{27}.cpm/6,0,[5,0,Welds2{27}.voltage,Welds2{27}.wfs,0,Welds2{27}.Current,0,0,0],[0,0,0,0,0,0,0,0,0]];
    wd28:=[Welds2{28}.cpm/6,0,[5,0,Welds2{28}.voltage,Welds2{28}.wfs,0,Welds2{28}.Current,0,0,0],[0,0,0,0,0,0,0,0,0]];
    wd29:=[Welds2{29}.cpm/6,0,[5,0,Welds2{29}.voltage,Welds2{29}.wfs,0,Welds2{29}.Current,0,0,0],[0,0,0,0,0,0,0,0,0]];
    wd30:=[Welds2{30}.cpm/6,0,[5,0,Welds2{30}.voltage,Welds2{30}.wfs,0,Welds2{30}.Current,0,0,0],[0,0,0,0,0,0,0,0,0]];
    wd31:=[Welds2{31}.cpm/6,0,[5,0,Welds2{31}.voltage,Welds2{31}.wfs,0,Welds2{31}.Current,0,0,0],[0,0,0,0,0,0,0,0,0]];
    wd32:=[Welds2{32}.cpm/6,0,[5,0,Welds2{32}.voltage,Welds2{32}.wfs,0,Welds2{32}.Current,0,0,0],[0,0,0,0,0,0,0,0,0]];
    wd33:=[Welds2{33}.cpm/6,0,[5,0,Welds2{33}.voltage,Welds2{33}.wfs,0,Welds2{33}.Current,0,0,0],[0,0,0,0,0,0,0,0,0]];
    wd34:=[Welds2{34}.cpm/6,0,[5,0,Welds2{34}.voltage,Welds2{34}.wfs,0,Welds2{34}.Current,0,0,0],[0,0,0,0,0,0,0,0,0]];
    wd35:=[Welds2{35}.cpm/6,0,[5,0,Welds2{35}.voltage,Welds2{35}.wfs,0,Welds2{35}.Current,0,0,0],[0,0,0,0,0,0,0,0,0]];
    wd36:=[Welds2{36}.cpm/6,0,[5,0,Welds2{36}.voltage,Welds2{36}.wfs,0,Welds2{36}.Current,0,0,0],[0,0,0,0,0,0,0,0,0]];
    wd37:=[Welds2{37}.cpm/6,0,[5,0,Welds2{37}.voltage,Welds2{37}.wfs,0,Welds2{37}.Current,0,0,0],[0,0,0,0,0,0,0,0,0]];
    wd38:=[Welds2{38}.cpm/6,0,[5,0,Welds2{38}.voltage,Welds2{38}.wfs,0,Welds2{38}.Current,0,0,0],[0,0,0,0,0,0,0,0,0]];
    wd39:=[Welds2{39}.cpm/6,0,[5,0,Welds2{39}.voltage,Welds2{39}.wfs,0,Welds2{39}.Current,0,0,0],[0,0,0,0,0,0,0,0,0]];
    wd40:=[Welds2{nMotionStepCount{2}}.cpm/6,0,[5,0,Welds2{nMotionStepCount{2}}.voltage,Welds2{nMotionStepCount{2}}.wfs,0,Welds2{nMotionStepCount{2}}.Current,0,0,0],[0,0,0,0,0,0,0,0,0]];

    Holdwd1:=[nHoldWeldVel,0,[5,0,Welds2{1}.voltage,Welds2{1}.wfs,0,Welds2{1}.Current,0,0,0],[0,0,0,0,0,0,0,0,0]];
    Holdwd2:=[nHoldWeldVel,0,[5,0,Welds2{2}.voltage,Welds2{2}.wfs,0,Welds2{2}.Current,0,0,0],[0,0,0,0,0,0,0,0,0]];
    Holdwd3:=[nHoldWeldVel,0,[5,0,Welds2{3}.voltage,Welds2{3}.wfs,0,Welds2{3}.Current,0,0,0],[0,0,0,0,0,0,0,0,0]];
    Holdwd4:=[nHoldWeldVel,0,[5,0,Welds2{4}.voltage,Welds2{4}.wfs,0,Welds2{4}.Current,0,0,0],[0,0,0,0,0,0,0,0,0]];
    Holdwd5:=[nHoldWeldVel,0,[5,0,Welds2{5}.voltage,Welds2{5}.wfs,0,Welds2{5}.Current,0,0,0],[0,0,0,0,0,0,0,0,0]];
    Holdwd6:=[nHoldWeldVel,0,[5,0,Welds2{6}.voltage,Welds2{6}.wfs,0,Welds2{6}.Current,0,0,0],[0,0,0,0,0,0,0,0,0]];
    Holdwd7:=[nHoldWeldVel,0,[5,0,Welds2{7}.voltage,Welds2{7}.wfs,0,Welds2{7}.Current,0,0,0],[0,0,0,0,0,0,0,0,0]];
    Holdwd8:=[nHoldWeldVel,0,[5,0,Welds2{8}.voltage,Welds2{8}.wfs,0,Welds2{8}.Current,0,0,0],[0,0,0,0,0,0,0,0,0]];
    Holdwd9:=[nHoldWeldVel,0,[5,0,Welds2{9}.voltage,Welds2{9}.wfs,0,Welds2{9}.Current,0,0,0],[0,0,0,0,0,0,0,0,0]];
    Holdwd10:=[nHoldWeldVel,0,[5,0,Welds2{10}.voltage,Welds2{10}.wfs,0,Welds2{10}.Current,0,0,0],[0,0,0,0,0,0,0,0,0]];

    ! --- Setup weave data (weave1..weave40) ---
    weave1:=[Welds2{1}.WeaveShape,Welds2{1}.WeaveType,Welds2{1}.WeaveLength,Welds2{1}.WeaveWidth,0,Welds2{1}.WeaveDwellLeft,0,Welds2{1}.WeaveDwellRight,0,0,0,0,0,0,0];
    weave2:=[Welds2{2}.WeaveShape,Welds2{2}.WeaveType,Welds2{2}.WeaveLength,Welds2{2}.WeaveWidth,0,Welds2{2}.WeaveDwellLeft,0,Welds2{2}.WeaveDwellRight,0,0,0,0,0,0,0];
    weave3:=[Welds2{3}.WeaveShape,Welds2{3}.WeaveType,Welds2{3}.WeaveLength,Welds2{3}.WeaveWidth,0,Welds2{3}.WeaveDwellLeft,0,Welds2{3}.WeaveDwellRight,0,0,0,0,0,0,0];
    weave4:=[Welds2{4}.WeaveShape,Welds2{4}.WeaveType,Welds2{4}.WeaveLength,Welds2{4}.WeaveWidth,0,Welds2{4}.WeaveDwellLeft,0,Welds2{4}.WeaveDwellRight,0,0,0,0,0,0,0];
    weave5:=[Welds2{5}.WeaveShape,Welds2{5}.WeaveType,Welds2{5}.WeaveLength,Welds2{5}.WeaveWidth,0,Welds2{5}.WeaveDwellLeft,0,Welds2{5}.WeaveDwellRight,0,0,0,0,0,0,0];
    weave6:=[Welds2{6}.WeaveShape,Welds2{6}.WeaveType,Welds2{6}.WeaveLength,Welds2{6}.WeaveWidth,0,Welds2{6}.WeaveDwellLeft,0,Welds2{6}.WeaveDwellRight,0,0,0,0,0,0,0];
    weave7:=[Welds2{7}.WeaveShape,Welds2{7}.WeaveType,Welds2{7}.WeaveLength,Welds2{7}.WeaveWidth,0,Welds2{7}.WeaveDwellLeft,0,Welds2{7}.WeaveDwellRight,0,0,0,0,0,0,0];
    weave8:=[Welds2{8}.WeaveShape,Welds2{8}.WeaveType,Welds2{8}.WeaveLength,Welds2{8}.WeaveWidth,0,Welds2{8}.WeaveDwellLeft,0,Welds2{8}.WeaveDwellRight,0,0,0,0,0,0,0];
    weave9:=[Welds2{9}.WeaveShape,Welds2{9}.WeaveType,Welds2{9}.WeaveLength,Welds2{9}.WeaveWidth,0,Welds2{9}.WeaveDwellLeft,0,Welds2{9}.WeaveDwellRight,0,0,0,0,0,0,0];
    weave10:=[Welds2{10}.WeaveShape,Welds2{10}.WeaveType,Welds2{10}.WeaveLength,Welds2{10}.WeaveWidth,0,Welds2{10}.WeaveDwellLeft,0,Welds2{10}.WeaveDwellRight,0,0,0,0,0,0,0];
    weave11:=[Welds2{11}.WeaveShape,Welds2{11}.WeaveType,Welds2{11}.WeaveLength,Welds2{11}.WeaveWidth,0,Welds2{11}.WeaveDwellLeft,0,Welds2{11}.WeaveDwellRight,0,0,0,0,0,0,0];
    weave12:=[Welds2{12}.WeaveShape,Welds2{12}.WeaveType,Welds2{12}.WeaveLength,Welds2{12}.WeaveWidth,0,Welds2{12}.WeaveDwellLeft,0,Welds2{12}.WeaveDwellRight,0,0,0,0,0,0,0];
    weave13:=[Welds2{13}.WeaveShape,Welds2{13}.WeaveType,Welds2{13}.WeaveLength,Welds2{13}.WeaveWidth,0,Welds2{13}.WeaveDwellLeft,0,Welds2{13}.WeaveDwellRight,0,0,0,0,0,0,0];
    weave14:=[Welds2{14}.WeaveShape,Welds2{14}.WeaveType,Welds2{14}.WeaveLength,Welds2{14}.WeaveWidth,0,Welds2{14}.WeaveDwellLeft,0,Welds2{14}.WeaveDwellRight,0,0,0,0,0,0,0];
    weave15:=[Welds2{15}.WeaveShape,Welds2{15}.WeaveType,Welds2{15}.WeaveLength,Welds2{15}.WeaveWidth,0,Welds2{15}.WeaveDwellLeft,0,Welds2{15}.WeaveDwellRight,0,0,0,0,0,0,0];
    weave16:=[Welds2{16}.WeaveShape,Welds2{16}.WeaveType,Welds2{16}.WeaveLength,Welds2{16}.WeaveWidth,0,Welds2{16}.WeaveDwellLeft,0,Welds2{16}.WeaveDwellRight,0,0,0,0,0,0,0];
    weave17:=[Welds2{17}.WeaveShape,Welds2{17}.WeaveType,Welds2{17}.WeaveLength,Welds2{17}.WeaveWidth,0,Welds2{17}.WeaveDwellLeft,0,Welds2{17}.WeaveDwellRight,0,0,0,0,0,0,0];
    weave18:=[Welds2{18}.WeaveShape,Welds2{18}.WeaveType,Welds2{18}.WeaveLength,Welds2{18}.WeaveWidth,0,Welds2{18}.WeaveDwellLeft,0,Welds2{18}.WeaveDwellRight,0,0,0,0,0,0,0];
    weave19:=[Welds2{19}.WeaveShape,Welds2{19}.WeaveType,Welds2{19}.WeaveLength,Welds2{19}.WeaveWidth,0,Welds2{19}.WeaveDwellLeft,0,Welds2{19}.WeaveDwellRight,0,0,0,0,0,0,0];
    weave20:=[Welds2{20}.WeaveShape,Welds2{20}.WeaveType,Welds2{20}.WeaveLength,Welds2{20}.WeaveWidth,0,Welds2{20}.WeaveDwellLeft,0,Welds2{20}.WeaveDwellRight,0,0,0,0,0,0,0];
    weave21:=[Welds2{21}.WeaveShape,Welds2{21}.WeaveType,Welds2{21}.WeaveLength,Welds2{21}.WeaveWidth,0,Welds2{21}.WeaveDwellLeft,0,Welds2{21}.WeaveDwellRight,0,0,0,0,0,0,0];
    weave22:=[Welds2{22}.WeaveShape,Welds2{22}.WeaveType,Welds2{22}.WeaveLength,Welds2{22}.WeaveWidth,0,Welds2{22}.WeaveDwellLeft,0,Welds2{22}.WeaveDwellRight,0,0,0,0,0,0,0];
    weave23:=[Welds2{23}.WeaveShape,Welds2{23}.WeaveType,Welds2{23}.WeaveLength,Welds2{23}.WeaveWidth,0,Welds2{23}.WeaveDwellLeft,0,Welds2{23}.WeaveDwellRight,0,0,0,0,0,0,0];
    weave24:=[Welds2{24}.WeaveShape,Welds2{24}.WeaveType,Welds2{24}.WeaveLength,Welds2{24}.WeaveWidth,0,Welds2{24}.WeaveDwellLeft,0,Welds2{24}.WeaveDwellRight,0,0,0,0,0,0,0];
    weave25:=[Welds2{25}.WeaveShape,Welds2{25}.WeaveType,Welds2{25}.WeaveLength,Welds2{25}.WeaveWidth,0,Welds2{25}.WeaveDwellLeft,0,Welds2{25}.WeaveDwellRight,0,0,0,0,0,0,0];
    weave26:=[Welds2{26}.WeaveShape,Welds2{26}.WeaveType,Welds2{26}.WeaveLength,Welds2{26}.WeaveWidth,0,Welds2{26}.WeaveDwellLeft,0,Welds2{26}.WeaveDwellRight,0,0,0,0,0,0,0];
    weave27:=[Welds2{27}.WeaveShape,Welds2{27}.WeaveType,Welds2{27}.WeaveLength,Welds2{27}.WeaveWidth,0,Welds2{27}.WeaveDwellLeft,0,Welds2{27}.WeaveDwellRight,0,0,0,0,0,0,0];
    weave28:=[Welds2{28}.WeaveShape,Welds2{28}.WeaveType,Welds2{28}.WeaveLength,Welds2{28}.WeaveWidth,0,Welds2{28}.WeaveDwellLeft,0,Welds2{28}.WeaveDwellRight,0,0,0,0,0,0,0];
    weave29:=[Welds2{29}.WeaveShape,Welds2{29}.WeaveType,Welds2{29}.WeaveLength,Welds2{29}.WeaveWidth,0,Welds2{29}.WeaveDwellLeft,0,Welds2{29}.WeaveDwellRight,0,0,0,0,0,0,0];
    weave30:=[Welds2{30}.WeaveShape,Welds2{30}.WeaveType,Welds2{30}.WeaveLength,Welds2{30}.WeaveWidth,0,Welds2{30}.WeaveDwellLeft,0,Welds2{30}.WeaveDwellRight,0,0,0,0,0,0,0];
    weave31:=[Welds2{31}.WeaveShape,Welds2{31}.WeaveType,Welds2{31}.WeaveLength,Welds2{31}.WeaveWidth,0,Welds2{31}.WeaveDwellLeft,0,Welds2{31}.WeaveDwellRight,0,0,0,0,0,0,0];
    weave32:=[Welds2{32}.WeaveShape,Welds2{32}.WeaveType,Welds2{32}.WeaveLength,Welds2{32}.WeaveWidth,0,Welds2{32}.WeaveDwellLeft,0,Welds2{32}.WeaveDwellRight,0,0,0,0,0,0,0];
    weave33:=[Welds2{33}.WeaveShape,Welds2{33}.WeaveType,Welds2{33}.WeaveLength,Welds2{33}.WeaveWidth,0,Welds2{33}.WeaveDwellLeft,0,Welds2{33}.WeaveDwellRight,0,0,0,0,0,0,0];
    weave34:=[Welds2{34}.WeaveShape,Welds2{34}.WeaveType,Welds2{34}.WeaveLength,Welds2{34}.WeaveWidth,0,Welds2{34}.WeaveDwellLeft,0,Welds2{34}.WeaveDwellRight,0,0,0,0,0,0,0];
    weave35:=[Welds2{35}.WeaveShape,Welds2{35}.WeaveType,Welds2{35}.WeaveLength,Welds2{35}.WeaveWidth,0,Welds2{35}.WeaveDwellLeft,0,Welds2{35}.WeaveDwellRight,0,0,0,0,0,0,0];
    weave36:=[Welds2{36}.WeaveShape,Welds2{36}.WeaveType,Welds2{36}.WeaveLength,Welds2{36}.WeaveWidth,0,Welds2{36}.WeaveDwellLeft,0,Welds2{36}.WeaveDwellRight,0,0,0,0,0,0,0];
    weave37:=[Welds2{37}.WeaveShape,Welds2{37}.WeaveType,Welds2{37}.WeaveLength,Welds2{37}.WeaveWidth,0,Welds2{37}.WeaveDwellLeft,0,Welds2{37}.WeaveDwellRight,0,0,0,0,0,0,0];
    weave38:=[Welds2{38}.WeaveShape,Welds2{38}.WeaveType,Welds2{38}.WeaveLength,Welds2{38}.WeaveWidth,0,Welds2{38}.WeaveDwellLeft,0,Welds2{38}.WeaveDwellRight,0,0,0,0,0,0,0];
    weave39:=[Welds2{39}.WeaveShape,Welds2{39}.WeaveType,Welds2{39}.WeaveLength,Welds2{39}.WeaveWidth,0,Welds2{39}.WeaveDwellLeft,0,Welds2{39}.WeaveDwellRight,0,0,0,0,0,0,0];
    weave40:=[Welds2{nMotionStepCount{2}}.WeaveShape,Welds2{nMotionStepCount{2}}.WeaveType,Welds2{nMotionStepCount{2}}.WeaveLength,Welds2{nMotionStepCount{2}}.WeaveWidth,0,Welds2{nMotionStepCount{2}}.WeaveDwellLeft,0,Welds2{nMotionStepCount{2}}.WeaveDwellRight,0,0,0,0,0,0,0];

    ! --- Compute vWeld speed array ---
    ! v3.5: Clamp minimum speed to 10mm/s to prevent ERRNO=205 (v_tcp=0 error)
    FOR i FROM 1 TO nMotionStepCount{2} DO
        nTempMmps:=Welds2{i}.cpm/6;
        IF nTempMmps < 0.1 nTempMmps:=10;
        vWeld{i}:=[nTempMmps,200,200,200];
    ENDFOR

    smDefault_2{1}.ign_move_delay:=2;
    Welds2{40}.position:=Welds2{nMotionStepCount{2}}.position;

    ! v3.5: Debug - log to file (nMotionStepCount, vWeld speeds, positions)
    jCurrent := CJointT();
    ! v3.12: Split to avoid ERR_STRTOOLNG (9E9 sentinel values = 10 digits)
    TPWrite "[R2_WELD] Gantry a="+NumToStr(jCurrent.extax.eax_a,0)+" b="+NumToStr(jCurrent.extax.eax_b,0);
    TPWrite "[R2_WELD] Gantry c="+NumToStr(jCurrent.extax.eax_c,0)+" d="+NumToStr(jCurrent.extax.eax_d,0);
    TPWrite "[R2_WELD] nMotionStepCount{2}="+NumToStr(nMotionStepCount{2},0);
    TPWrite "[R2_WELD] Welds2{1}.pos=["+NumToStr(Welds2{1}.position.trans.x,1)+","+NumToStr(Welds2{1}.position.trans.y,1)+","+NumToStr(Welds2{1}.position.trans.z,1)+"] conf=["+NumToStr(Welds2{1}.position.robconf.cf1,0)+","+NumToStr(Welds2{1}.position.robconf.cf4,0)+"]";
    TPWrite "[R2_WELD] wobjWeldLine2.uframe=["+NumToStr(wobjWeldLine2.uframe.trans.x,1)+","+NumToStr(wobjWeldLine2.uframe.trans.y,1)+","+NumToStr(wobjWeldLine2.uframe.trans.z,1)+"]";
    ! v3.6: Write startup info to existing error log (no new file = no ERRNO=205)
    ! Note: robot2_weld_error.txt already exists from previous runs, \Append is safe
    Open "HOME:/robot2_weld_error.txt", weld2_errlog \Append;
    Write weld2_errlog, "=== v3.12 START " + CTime() + " nMotionStepCount=" + NumToStr(nMotionStepCount{2},0) + " nMotionStartStepLast=" + NumToStr(nMotionStartStepLast{2},0) + " ===";
    Close weld2_errlog;
    nErrorCount := 0;
    nMotionErrorCount := 0;

    ! v4.0: Correct gantry-traversal architecture
    ! Phase 1: Robot arm moves 0->50mm  (Welds2{1}->{2}, gantry stopped)
    ! Phase 2: Robot holds/oscillates   (Welds2{2}<->{3}, gantry traverses 50->950mm)
    ! Phase 3: Robot arm final          (Welds2{3}, gantry stopped at 950mm)
    ! Sync: WaitUntil t1_weld_start (begin), WHILE NOT t1_weld_done (hold end)
    ConfJ\Off;
    ConfL\Off;
    WaitRob\ZeroSpeed;

    ! Wait for TASK1 TraceWeldLine to start
    TPWrite "[R2_WELD] Waiting for t1_weld_start...";
    WaitUntil t1_weld_start = TRUE;
    TPWrite "[R2_WELD] t1_weld_start received - begin arc";

    ! ===== Phase 1: Robot arm 0->50mm =====
    nRunningStep{2} := 1;
    TPWrite "[R2_WELD] Phase1: MoveJ Welds2{1} (weld start approach)";
    MoveJ Welds2{1}.position, vTargetSpeed, fine, tWeld2\WObj:=wobjWeldLine2;

    nRunningStep{2} := 2;
    TPWrite "[R2_WELD] Phase1: MoveL Welds2{2} (0->50mm robot arc)";
    MoveL Welds2{2}.position, vWeld{2}, fine, tWeld2\WObj:=wobjWeldLine2;

    ! ===== Phase 2: Wait for gantry traversal (WaitUntil - no oscillation until Welds2 re-taught) =====
    nRunningStep{2} := 3;
    TPWrite "[R2_WELD] Phase2: WaitUntil t1_weld_done (gantry traversing 50->950mm)";
    WaitUntil t1_weld_done = TRUE;
    TPWrite "[R2_WELD] Phase2: t1_weld_done received";

    ! ===== Phase 3: Final position =====
    nRunningStep{2} := 4;
    TPWrite "[R2_WELD] Phase3: MoveL Welds2{3} (final)";
    MoveL Welds2{3}.position, vWeld{3}, fine, tWeld2\WObj:=wobjWeldLine2;

    ! Done
    ConfL\On;
    ConfJ\On;
    TPWrite "[R2_WELD] Robot2_EdgeWeldSequence v4.0 done";
ERROR
    ! 50050: Welds2 position outside reach - skip until re-teaching done
    IF ERRNO = 50050 THEN
        TPWrite "[R2_WELD] SKIP50050 step=" + NumToStr(nRunningStep{2},0) + " (re-teaching needed)";
        TRYNEXT;
    ENDIF
    TPWrite "[R2_WELD] ERROR ERRNO=" + NumToStr(ERRNO,0) + " step=" + NumToStr(nRunningStep{2},0);
    ConfL\On;
    ConfJ\On;
ENDPROC


! ========================================
! Command Loop (v2.1.0 - PlanA Style)
! ========================================
! Robot2 command monitoring loop
! Responds to nCmdInput changes from upper system

! ----------------------------------------
! Robot2_CommandLoop: Command monitoring loop
! ----------------------------------------
! Monitors nCmdInput and executes Robot2-specific actions
PROC Robot2_CommandLoop()
	VAR num last_cmd := 0;

	TPWrite "========================================";
	TPWrite "[R2_CMD] Entering Command Loop (v2.1.0)";
	TPWrite "[R2_CMD] Monitoring nCmdInput...";
	TPWrite "========================================";

	WHILE TRUE DO
		! Wait for new command from upper system
		WaitUntil nCmdInput <> 0 AND nCmdInput <> last_cmd;
		last_cmd := nCmdInput;

		TPWrite "[R2_CMD] Command received: " + NumToStr(nCmdInput, 0);

		TEST nCmdInput
		CASE CMD_MOVE_TO_WORLDHOME:
			TPWrite "[R2_CMD] Move to World Home";
			SetRobot2InitialPosition;

		CASE CMD_WELD, CMD_WELD_MOTION:
			TPWrite "[R2_CMD] Weld Sequence";
			Robot2_WeldSequence;

		CASE CMD_EDGE_WELD:
			TPWrite "[R2_CMD] Edge-based Weld";
			Robot2_EdgeWeldSequence;

		CASE CMD_ROB2_WIRE_CUT:
			TPWrite "[R2_CMD] Robot2 Wire Cut";
			! TODO: Implement wire cut

		DEFAULT:
			! Non-Robot2 specific commands - just wait
			TPWrite "[R2_CMD] Waiting (cmd=" + NumToStr(nCmdInput, 0) + ")";

		ENDTEST

		! Wait for command to be cleared
		WaitUntil nCmdInput = 0;
		last_cmd := 0;

		TPWrite "[R2_CMD] Ready for next command";
	ENDWHILE
ENDPROC

! ========================================
! Rob2_CommandListener: T_Head stCommand handler (v1.9.43)
! ========================================
! Responds to stCommand from T_Head task
! Protocol: "Ready" -> receive command -> execute -> "Ack" -> wait clear -> "Ready"
PROC Rob2_CommandListener()
	VAR iodev head_log;
	Open "HOME:/head_r2_listener.txt", head_log \Write;
	Write head_log, "Rob2 CommandListener (v1.9.43) - " + CDate() + " " + CTime();

	TPWrite "[R2] CommandListener started, entering Ready state";

	WHILE TRUE DO
		stReact{2} := "Ready";
		Write head_log, "Status: Ready, waiting stCommand...";
		WaitUntil stCommand <> "";
		Write head_log, "Received: " + stCommand;
		TPWrite "[R2] stCommand=" + stCommand;

		TEST stCommand
			CASE "MoveHome":
				stReact{2} := "";
				SetRobot2InitialPosition;
				stReact{2} := "Ack";
				Write head_log, "MoveHome done";
				WaitUntil stCommand = "";

			CASE "MoveJgJ":
				stReact{2} := "";
				! v1.9.44: Move Robot2 to target joint position from T_Head
				MoveAbsJ jRob2, vSync, fine, tool0;
				stReact{2} := "Ack";
				Write head_log, "MoveJgJ done";
				WaitUntil stCommand = "";

			CASE "MovePgJ":
				stReact{2} := "";
				MoveJ pRob2, vSync, zSync, tool0;
				stReact{2} := "Ack";
				Write head_log, "MovePgJ done";
				WaitUntil stCommand = "";

			CASE "MovePgL":
				stReact{2} := "";
				MoveL pRob2, vSync, zSync, tool0;
				stReact{2} := "Ack";
				Write head_log, "MovePgL done";
				WaitUntil stCommand = "";

			CASE "EdgeWeld":
				stReact{2} := "";
				Write head_log, "EdgeWeld: waiting t1_weld_position_ready";
				WaitUntil t1_weld_position_ready = TRUE \MaxTime := 60;
				IF t1_weld_position_ready THEN
					Robot2_EdgeWeldSequence;
					WaitUntil t1_weld_done = TRUE \MaxTime := 120;
				ELSE
					Write head_log, "EdgeWeld: t1_weld_position_ready timeout";
					TPWrite "[R2] ERROR: t1_weld_position_ready timeout";
				ENDIF
				stReact{2} := "Ack";
				Write head_log, "EdgeWeld done";
				WaitUntil stCommand = "";

			CASE "Weld", "WeldMotion", "WeldCorr", "WeldMotionCorr":
				stReact{2} := "";
				Write head_log, "Weld: waiting t1_weld_position_ready";
				WaitUntil t1_weld_position_ready = TRUE \MaxTime := 60;
				IF t1_weld_position_ready THEN
					Robot2_EdgeWeldSequence;
					WaitUntil t1_weld_done = TRUE \MaxTime := 120;
				ELSE
					Write head_log, "Weld: t1_weld_position_ready timeout";
					TPWrite "[R2] ERROR: t1_weld_position_ready timeout";
				ENDIF
				stReact{2} := "Ack";
				Write head_log, "Weld done";
				WaitUntil stCommand = "";

			CASE "Rob2WireCut":
				stReact{2} := "";
				! Stub - Robot2 wire cut
				stReact{2} := "Ack";
				Write head_log, "Rob2WireCut done (stub)";
				WaitUntil stCommand = "";

			CASE "checkpos":
				stReact{2} := "";
				rT_ROB2check;
				stReact{2} := "checkposok";
				Write head_log, "checkpos done";
				WaitUntil stCommand = "";

			DEFAULT:
				! TASK1-only commands (MoveAbsGantry, TestMenu etc.)
				! Robot2 not involved - immediate Ack
				! Note: rDispatchR1 is used for these, so this rarely triggers
				Write head_log, "Not R2 command: " + stCommand + " (immediate Ack)";
				stReact{2} := "Ack";
				WaitUntil stCommand = "";
		ENDTEST
	ENDWHILE
ERROR
	Write head_log, "ERROR " + NumToStr(ERRNO, 0);
	Close head_log;
ENDPROC

    ! ========================================
    ! fCalcWeldingpos: Welding position interpolation
    ! ========================================
    ! Ported from PlanA T_ROB2_Function.mod
    ! Computes next interpolated position along weld path (0.5mm step)
    FUNC robtarget fCalcWeldingpos(robtarget CurrentPos,robtarget Start,robtarget End)
        VAR robtarget result;
        VAR robtarget pCalcTemp;
        VAR num nCalcCount;
        nCalcCount:=round(VectMagn(End.trans-Start.trans)/0.5);
        pCalcTemp.trans:=(End.trans-Start.trans)/nCalcCount;
        tool_rx_end:=[EulerZYX(\z,End.rot),EulerZYX(\y,End.rot),EulerZYX(\x,End.rot)];
        tool_rx_start:=[EulerZYX(\z,Start.rot),EulerZYX(\y,Start.rot),EulerZYX(\x,Start.rot)];
        tool_rx_delta:=[(tool_rx_end{1}-tool_rx_start{1})/nCalcCount,(tool_rx_end{2}-tool_rx_start{2})/nCalcCount,(tool_rx_end{3}-tool_rx_start{3})/nCalcCount];
        result.trans:=CurrentPos.trans+pCalcTemp.trans;
        result.rot:=(OrientZYX(EulerZYX(\z,CurrentPos.rot)+tool_rx_delta{1},EulerZYX(\y,CurrentPos.rot)+tool_rx_delta{2},EulerZYX(\x,CurrentPos.rot)));
        result.extax:=[9e9,9e9,9e9,9e9,9e9,9e9];
        RETURN result;
    ENDFUNC

ENDMODULE
